// TIA Portal V15.1 export
// export: Created 2026-01-09T13:45:11.7129473Z, ExportSetting WithDefaults, WithReadOnly, DisplayName Totally Integrated Automation Portal, DisplayVersion V15.1 Update 8, DisplayName TIA Portal Openness, DisplayVersion V15.1 Update 8, DisplayName STEP 7 Professional, DisplayVersion V15.1 Update 8, DisplayName WinCC Advanced, DisplayVersion V15.1 Update 8
DATA_BLOCK "C#5_WD_TIMER"   // DB5
{ S7_Optimized_Access := 'FALSE' }
VERSION : 0.1
// stored: AutoNumber true, CodeModifiedDate 2024-09-25T16:11:16.0895396Z, CompileDate 2025-08-30T17:40:34.4162196Z, CreationDate 2024-10-12T12:36:08.0193576Z, DBAccessibleFromOPCUA true, InterfaceModifiedDate 2024-09-25T16:11:16.0895396Z, IsConsistent true, IsKnowHowProtected false, IsOnlyStoredInLoadMemory false, IsPLCDB false, IsWriteProtectedInAS false, ModifiedDate 2024-10-13T07:10:46.0630795Z, ParameterModified 2024-09-25T16:11:16.0895396Z, StructureModified 2024-09-25T16:11:16.0895396Z
   VAR RETAIN
      TG_Tron : Real;   // Thời gian trộn
      TG_Xa100 : Real;   // Thời gian mở cửa nồi 100
      "TG_Xa FD Sau AG" : Real;   // Thời gian xả FD sau AG
      "TG_Xa AP Sau AG" : Real;   // Thời gian xả AP sau AG
      "TG_Xa SBS Sau AG" : Real;   // Thời gian xả SBS sau AG
      "TG_Bom Tuoi Nhua" : Real;   // Thời gian bơm tưới nhựa chạy thêm
      HSN_AG1 : Real;   // Hệ số nạp mô phỏng AG1
      HSN_AG2 : Real;   // Hệ số nạp mô phỏng AG2
      HSN_AG3 : Real;   // Hệ số nạp mô phỏng AG3
      HSN_AG4 : Real;   // Hệ số nạp mô phỏng AG4
      HSN_AG5 : Real;   // Hệ số nạp mô phỏng AG5
      HSX_AG1 : Real;   // Hệ số xả mô phỏng AG1
      HSN_FD1 : Real;   // Hệ số nạp mô phỏng FD1
      HSX_FD1 : Real;   // Hệ số xả mô phỏng FD1
      HSN_AP1 : Real;   // Hệ số nạp mô phỏng AP1
      HSX_AP1 : Real;   // Hệ số xả mô phỏng AP1
      HSN_SB1 : Real;   // Hệ số nạp mô phỏng SBS1
      HSX_SB1 : Real;   // Hệ số xả mô phỏng SBS1
   END_VAR
BEGIN
END_DATA_BLOCK
